INTERFACE IGHT

{attribute 'object_name' := 'AddItem'}
METHOD AddItem : BOOL
VAR_INPUT
	uliKey: ULINT;
	pData: POINTER TO BYTE;
END_VAR
END_METHOD

PROPERTY Count : UINT
GET
END_GET
END_PROPERTY

{attribute 'object_name' := 'Lookup'}
METHOD Lookup : POINTER TO BYTE
VAR_INPUT
	uliKey: ULINT;
	bolRemove: BOOL;
END_VAR
END_METHOD

{attribute 'object_name' := 'Clear'}
METHOD Clear : BOOL
VAR_INPUT
	bolFreePointer: BOOL;
END_VAR
END_METHOD

{attribute 'object_name' := 'Initialize'}
METHOD Initialize : BOOL
END_METHOD

END_INTERFACE

(* stored: Version 1.1.0.1, ProductVersion 3.1.0.36
   Itf IGHT: Id {8288fcde-3df1-4b79-a15a-f2022929c3f5}
   Method AddItem: Id {03bcbad2-cfa3-41c9-a1e4-ef37900c3322}
   Property Count: Id {0513c588-335d-4f9b-a9b0-d5af1f916936}
   Get Get: Id {6ad5dc3c-4923-4790-97f3-a8f71db02614}
   Method Lookup: Id {39a17a39-6291-41c5-8c81-f2e3156499d5}
   Method Clear: Id {e01acbdd-b6df-460a-ac1e-c0e9c118f2d3}
   Method Initialize: Id {e4dd3a6d-7673-45c1-b425-39c063309288} *)
